FUNCTION_BLOCK FlowController (* Composite Function Block Type *)
  (* Standard: 61499-2 *)
  (* Version 0.0, 2011-12-18, 4DIAC-IDE, 4DIAC-Consortium *)
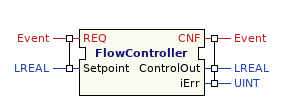
  EVENT_INPUT
    REQ WITH Setpoint; (* Normal Execution Request *)
  END_EVENT
  EVENT_OUTPUT
    CNF WITH ControlOut, iErr; (* Execution Confirmation *)
  END_EVENT
  VAR_INPUT
    Setpoint : LREAL; (* Input event qualifier *)
  END_VAR
  VAR_OUTPUT
    ControlOut : LREAL; (* Output event qualifier *)
    iErr : UINT;
  END_VAR
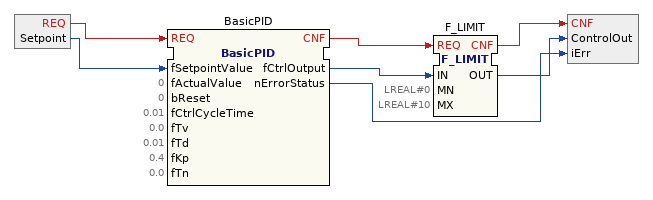
  FBS
    BasicPID : BasicPID(fActualValue := 0, bReset := 0, fCtrlCycleTime := 0.01, fTv := 0.0, fTd := 0.01, fKp := 0.4, fTn := 0.0);
    F_LIMIT : F_LIMIT(MN := LREAL#0, MX := LREAL#10);
  END_FBS
  EVENT_CONNECTIONS
    REQ TO BasicPID.REQ;
    F_LIMIT.CNF TO CNF;
    BasicPID.CNF TO F_LIMIT.REQ;
  END_CONNECTIONS
  DATA_CONNECTIONS
    Setpoint TO BasicPID.fSetpointValue;
    BasicPID.nErrorStatus TO iErr;
    BasicPID.fCtrlOutput TO F_LIMIT.IN;
    F_LIMIT.OUT TO ControlOut;
  END_CONNECTIONS
END_FUNCTION_BLOCK
